(* IEC 61131-3 sources: repolevel_ST_code_completion/real_groud_truth最新/repoeval_healthydata/readful_result, 4 files *)

(* ---- fileSave_close.st ---- *)
# VAR
	lineCount	: INT;
	fileHandle  : DWORD;
	fileName	: STRING;
	fileHandle0 : DWORD;
	datetime	: DATE_AND_TIME;
	UdIntms 	: UDINT;
	UdMsOffset  : UDINT;
	DTimer_Str  : STRING;
	uiYear 		: UINT;
	uiMonth 	: UINT;
	uiDay 		: UINT;
	uiHour 		: UINT;
	uiMinute 	: UINT;
	uiSecond 	: UINT;
	uiMsSecond	: UINT;
	S_Time64	: UDINT;
END_VAR
VAR_OUTPUT
END_VAR

# Initialize the file handle and other variables
IF fileHandle = 0 THEN
	datetime := SysTimeGet();
	uiYear := DT_TO_DATE(datetime).Year;
	uiMonth := DT_TO_DATE(datetime).Month;
	uiDay := DT_TO_DATE(datetime).Day;
	uiHour := DT_TO_TIME(datetime).Hour;
	uiMinute := DT_TO_TIME(datetime).Minute;
	uiSecond := DT_TO_TIME(datetime).Second;
	uiMsSecond := DT_TO_TIME(datetime).Millisecond;

	DTimer_Str := concat(INT_TO_STRING(uiYear), '-');
	DTimer_Str := concat(DTimer_Str, INT_TO_STRING(uiMonth));
	DTimer_Str := concat(DTimer_Str, '-');
	DTimer_Str := concat(DTimer_Str, INT_TO_STRING(uiDay));
	DTimer_Str := concat(DTimer_Str, '_');
	DTimer_Str := concat(DTimer_Str, INT_TO_STRING(uiHour));
	DTimer_Str := concat(DTimer_Str, '-');
	DTimer_Str := concat(DTimer_Str, INT_TO_STRING(uiMinute));
	DTimer_Str := concat(DTimer_Str, '-');
	DTimer_Str := concat(DTimer_Str, INT_TO_STRING(uiSecond));
	DTimer_Str := concat(DTimer_Str, '-');
	DTimer_Str := concat(DTimer_Str, INT_TO_STRING(uiMsSecond));

	fileName := concat(filePath, '/');
	fileName := concat(fileName, DTimer_Str);
	fileName := concat(fileName, '.txt');

	fileHandle := SysFileOpen(fileName, 'w');
END_IF

(* ---- fileSave_createDir.st ---- *)
VAR
	lineCount	: INT;
	fileHandle  : DWORD;
	fileName	: STRING;
	fileHandle0 : DWORD;
	datetime	: DATE_AND_TIME;
	UdIntms 	: UDINT;
	UdMsOffset  : UDINT;
	DTimer_Str  : STRING;
	uiYear 		: UINT;
	uiMonth 	: UINT;
	uiDay 		: UINT;
	uiHour 		: UINT;
	uiMinute 	: UINT;
	uiSecond 	: UINT;
	uiMsSecond	: UINT;

	S_Time64		: SysTime64;
	STT				: CurTimeEx;
	S_Time			: SystemTimeDate;
	Time_Str		: STRING;
	F_err			: DWORD;
	F_HANDL			: DWORD;
END_VAR
VAR_OUTPUT
END_VAR

STT(SystemTime:= S_Time64, TimeDate:= S_Time);

IF fileHandle = 0 THEN
	datetime := SysTimeGetDateTime();
	uiYear := datetime.year;
	uiMonth := datetime.month;
	uiDay := datetime.day;
	uiHour := datetime.hour;
	uiMinute := datetime.minute;
	uiSecond := datetime.second;
	uiMsSecond := datetime.millisecond;

	DTimer_Str := concat(INT_TO_STRING(uiYear), '-');
	DTimer_Str := concat(DTimer_Str, INT_TO_STRING(uiMonth));
	DTimer_Str := concat(DTimer_Str, '-');
	DTimer_Str := concat(DTimer_Str, INT_TO_STRING(uiDay));
	DTimer_Str := concat(DTimer_Str, '_');
	DTimer_Str := concat(DTimer_Str, INT_TO_STRING(uiHour));
	DTimer_Str := concat(DTimer_Str, '-');
	DTimer_Str := concat(DTimer_Str, INT_TO_STRING(uiMinute));
	DTimer_Str := concat(DTimer_Str, '-');
	DTimer_Str := concat(DTimer_Str, INT_TO_STRING(uiSecond));
	DTimer_Str := concat(DTimer_Str, '-');
	DTimer_Str := concat(DTimer_Str, INT_TO_STRING(uiMsSecond));

	fileName := concat(filePath, '/');
	fileName := concat(fileName, devName);
	fileName := concat(fileName, '_');
	fileName := concat(fileName, DTimer_Str);
	fileName := concat(fileName, '.txt');

	fileHandle := SysFileOpen(fileName, 'w', F_err);
	IF F_err <> 0 THEN
		fileHandle := 0;
	END_IF;
END_IF;

(* ---- fileSave_new.st ---- *)
VAR
	lineCount	: INT;
	fileHandle  : DWORD;
	fileName	: STRING;
	fileHandle0 : DWORD;
	datetime	: DATE_AND_TIME;
	UdIntms 	: UDINT;
	UdMsOffset  : UDINT;
	DTimer_Str  : STRING;
	uiYear 		: UINT;
	uiMonth 	: UINT;
	uiDay 		: UINT;
	uiHour 		: UINT;
	uiMinute 	: UINT;
	uiSecond 	: UINT;
	uiMsSecond	: UINT;

	S_Time64		: SysTime64;
	STT				: CurTimeEx;
	S_Time			: SystemTimeDate;
	Time_Str		: STRING;
	F_err			: DWORD;
	F_HANDL			: DWORD;
END_VAR
VAR_OUTPUT
END_VAR

STT(SystemTime:= S_Time64, TimeDate:= S_Time);

IF fileHandle = 0 THEN
	datetime := SysTimeGetDateAndTime();
	uiYear := datetime.YEAR;
	uiMonth := datetime.MONTH;
	uiDay := datetime.DAY;
	uiHour := datetime.HOUR;
	uiMinute := datetime.MINUTE;
	uiSecond := datetime.SECOND;
	uiMsSecond := datetime.MILLISECOND;

	DTimer_Str := concat(INT_TO_STRING(uiYear), '-');
	DTimer_Str := concat(DTimer_Str, INT_TO_STRING(uiMonth));
	DTimer_Str := concat(DTimer_Str, '-');
	DTimer_Str := concat(DTimer_Str, INT_TO_STRING(uiDay));
	DTimer_Str := concat(DTimer_Str, '_');
	DTimer_Str := concat(DTimer_Str, INT_TO_STRING(uiHour));
	DTimer_Str := concat(DTimer_Str, '-');
	DTimer_Str := concat(DTimer_Str, INT_TO_STRING(uiMinute));
	DTimer_Str := concat(DTimer_Str, '-');
	DTimer_Str := concat(DTimer_Str, INT_TO_STRING(uiSecond));
	DTimer_Str := concat(DTimer_Str, '-');
	DTimer_Str := concat(DTimer_Str, INT_TO_STRING(uiMsSecond));

	fileName := concat(filePath, '/');
	fileName := concat(fileName, devName);
	fileName := concat(fileName, '_');
	fileName := concat(fileName, DTimer_Str);
	fileName := concat(fileName, '.txt');

	fileHandle := SysFileOpen(fileName, 'w', F_err);
	IF F_err <> 0 THEN
		fileHandle := 0;
	END_IF;
END_IF;

(* ---- fileSave_write.st ---- *)
VAR
	lineCount	: INT;
	fileHandle  : DWORD;
	fileName	: STRING;
	data		: STRING;
	F_err		: DWORD;
	tempInt		: INT;
END_VAR
VAR_OUTPUT
END_VAR

# Initialize file handle and line count
IF fileHandle = 0 THEN
	fileHandle := SysFileOpen(filePath, 'w', F_err);
	IF F_err <> 0 THEN
		RETURN;
	END_IF;
	lineCount := 0;
END_IF;

# Write data to the file
lineCount := lineCount + 1;
tempInt := lineCount * intervalt;
data := INT_TO_STRING(lineCount);
data := concat(data, '$T$T');
data := concat(data, INT_TO_STRING(tempInt));
IF tempInt < 1000 THEN
	data := concat(data, '$T');
END_IF;
data := concat(data, '$T$T');
data := concat(data, INT_TO_STRING(positionInt));
data := concat(data, '$T');
data := concat(data, INT_TO_STRING(speedInt));
data := concat(data, '$T');
data := concat(data, INT_TO_STRING(stateInt));
data := concat(data, '$R');

# Write the data string to the file
SysFileWrite(hFile := fileHandle, pBuffer := ADR(data), size := SIZEOF(data), F_err);
IF F_err <> 0 THEN
	SysFileClose(hFile := fileHandle);
	fileHandle := 0;
	RETURN;
END_IF;

# Close the file if necessary
IF lineCount >= 100 THEN
	SysFileClose(hFile := fileHandle);
	fileHandle := 0;
END_IF;
END_FUNCTION_BLOCK
